FUNCTION_BLOCK AsyncEchoRpcHandler IMPLEMENTS I_RpcHandler
VAR
	asyncResponse : I_AsynchronousRpcResponse;
	result : T_MAXSTRING;
	timer : TON;
END_VAR

PROPERTY PUBLIC Busy : BOOL
GET
Busy := asyncResponse <> 0;
END_GET
END_PROPERTY

METHOD PUBLIC CyclicCall
VAR_INPUT
END_VAR
timer(in := Busy, pt := T#1S);

IF timer.Q THEN
	asyncResponse.CompleteWithString(result);
	asyncResponse.Dispose();
	asyncResponse := 0;
	result := '';
END_IF
END_METHOD

METHOD Handle
VAR_INPUT
	Parameters : I_Deserializer;
	Response : I_SynchronousRpcResponse;
END_VAR
VAR
	echo : T_MAXSTRING;
END_VAR
IF Busy THEN
	Response.RejectWithMessage('Already processing response');
	RETURN;
END_IF

IF NOT Parameters.TryGetKeyString('Echo',echo) THEN
	Response.RejectWithMessage('Missing Echo parameter');
	RETURN;
END_IF

result := echo;
Response.TryMakeAsynchronous(asyncResponse);
END_METHOD

END_FUNCTION_BLOCK

(* stored: Version 1.1.0.1, ProductVersion 3.1.4024.12
   POU AsyncEchoRpcHandler: Id {1e2412a2-f1b1-4465-80c2-0a0e7fcc5168}, SpecialFunc None
   Property Busy: Id {e084576c-3d84-48ad-b478-14feb8f6ed04}
   Get Get: Id {94ca94e5-a0e8-4bd8-b5a5-21e7b7ae0091}
   Method CyclicCall: Id {600e73b5-f953-4466-967d-a80822e095b2}
   Method Handle: Id {85791512-73b6-4c83-9c38-6e85292f49d0} *)
